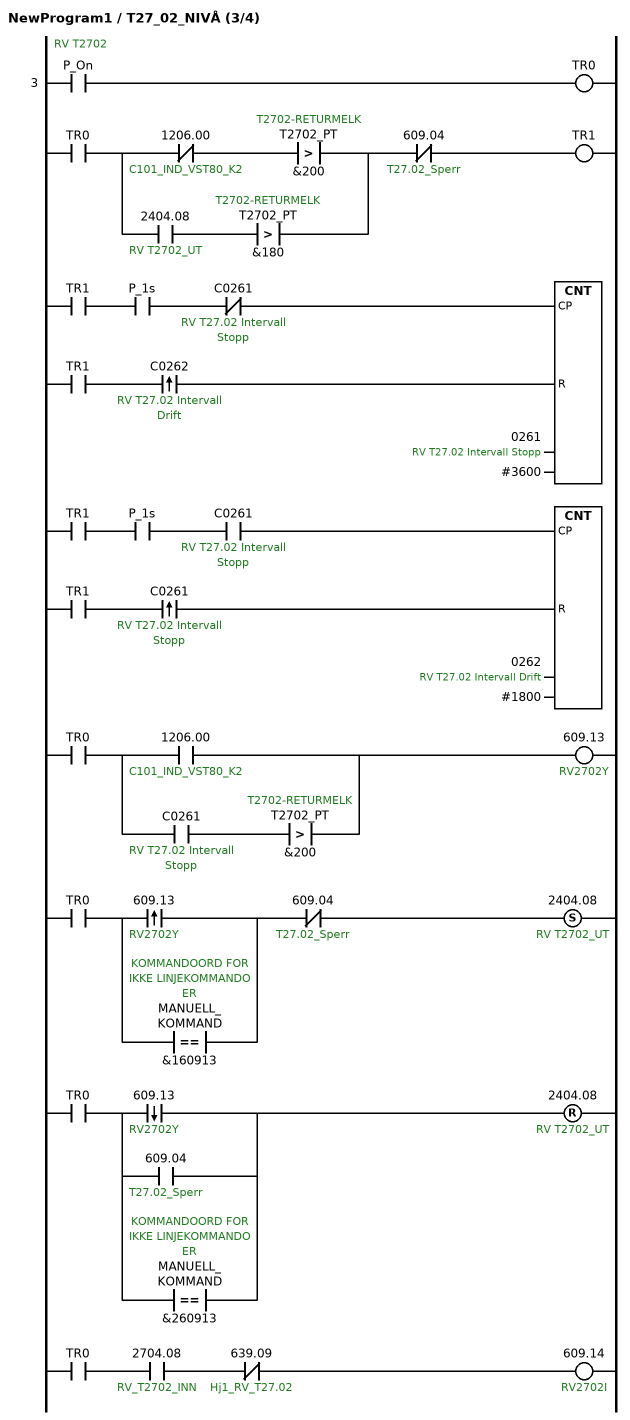
; [picture p984: NewProgram1 / T27_02_NIVÅ, rungs 3-3]
; rung 3: RV T2702
LD P_On
OUT TR0
LDNOT 1206.00  ; C101_IND_VST80_K2
AND>(320) T2702_PT &200  ; T2702-RETURMELK
LD 2404.08  ; RV T2702_UT
AND>(320) T2702_PT &180  ; T2702-RETURMELK
ORLD
ANDLD
ANDNOT 609.04  ; T27.02_Sperr
OUT TR1
AND P_1s
ANDNOT C0261  ; RV T27.02 Intervall Stopp
LD TR1
@AND C0262  ; RV T27.02 Intervall Drift
CNT 0261 #3600  ; RV T27.02 Intervall Stopp
LD TR1
AND P_1s
AND C0261  ; RV T27.02 Intervall Stopp
LD TR1
@AND C0261  ; RV T27.02 Intervall Stopp
CNT 0262 #1800  ; RV T27.02 Intervall Drift
LD TR0
LD 1206.00  ; C101_IND_VST80_K2
LD C0261  ; RV T27.02 Intervall Stopp
AND>(320) T2702_PT &200  ; T2702-RETURMELK
ORLD
ANDLD
OUT 609.13  ; RV2702Y
LD TR0
@LD 609.13  ; RV2702Y
OR=L(301) MANUELL_KOMMAND &160913  ; KOMMANDOORD FOR IKKE LINJEKOMMANDOER
ANDLD
ANDNOT 609.04  ; T27.02_Sperr
SET 2404.08  ; RV T2702_UT
LD TR0
%LD 609.13  ; RV2702Y
OR 609.04  ; T27.02_Sperr
OR=L(301) MANUELL_KOMMAND &260913  ; KOMMANDOORD FOR IKKE LINJEKOMMANDOER
ANDLD
RSET 2404.08  ; RV T2702_UT
LD TR0
AND 2704.08  ; RV_T2702_INN
ANDNOT 639.09  ; Hj1_RV_T27.02
OUT 609.14  ; RV2702I

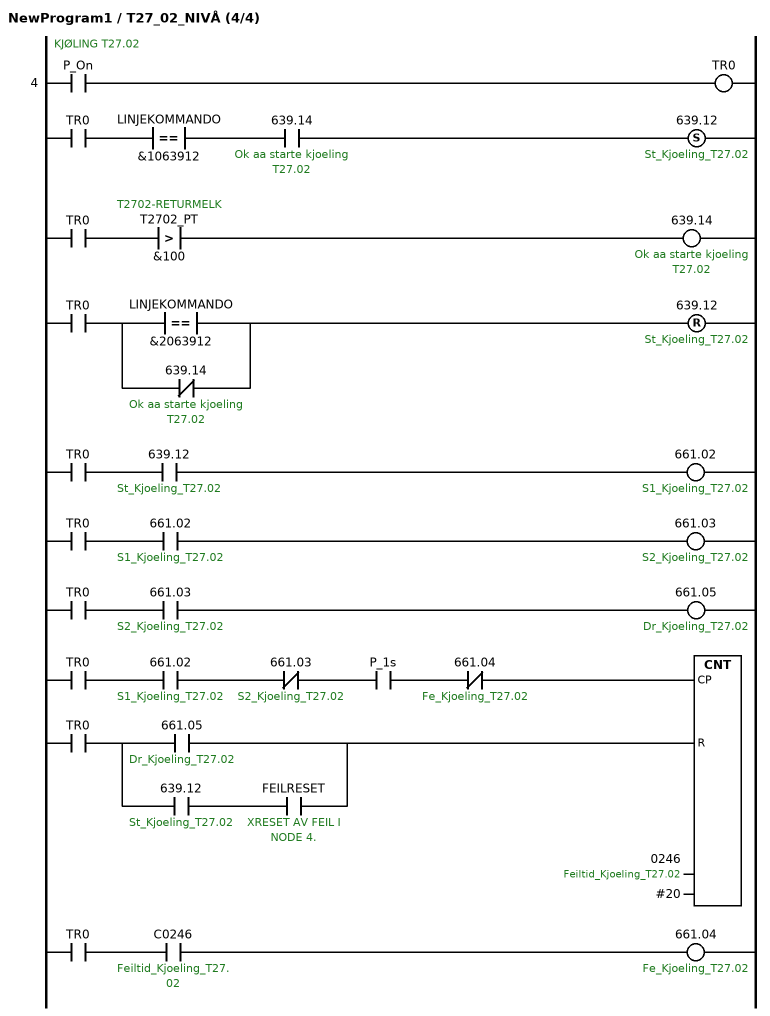
; rung 4: KJØLING T27.02
LD P_On
OUT TR0
AND=L(301) LINJEKOMMANDO &1063912
AND 639.14  ; Ok aa starte kjoeling T27.02
SET 639.12  ; St_Kjoeling_T27.02
LD TR0
AND>(320) T2702_PT &100  ; T2702-RETURMELK
OUT 639.14  ; Ok aa starte kjoeling T27.02
LD TR0
LD=L(301) LINJEKOMMANDO &2063912
ORNOT 639.14  ; Ok aa starte kjoeling T27.02
ANDLD
RSET 639.12  ; St_Kjoeling_T27.02
LD TR0
AND 639.12  ; St_Kjoeling_T27.02
OUT 661.02  ; S1_Kjoeling_T27.02
LD TR0
AND 661.02  ; S1_Kjoeling_T27.02
OUT 661.03  ; S2_Kjoeling_T27.02
LD TR0
AND 661.03  ; S2_Kjoeling_T27.02
OUT 661.05  ; Dr_Kjoeling_T27.02
LD TR0
AND 661.02  ; S1_Kjoeling_T27.02
ANDNOT 661.03  ; S2_Kjoeling_T27.02
AND P_1s
ANDNOT 661.04  ; Fe_Kjoeling_T27.02
LD TR0
LD 661.05  ; Dr_Kjoeling_T27.02
LD 639.12  ; St_Kjoeling_T27.02
AND FEILRESET  ; XRESET AV FEIL I NODE 4.
ORLD
ANDLD
CNT 0246 #20  ; Feiltid_Kjoeling_T27.02
LD TR0
AND C0246  ; Feiltid_Kjoeling_T27.02
OUT 661.04  ; Fe_Kjoeling_T27.02

### Section T27_02

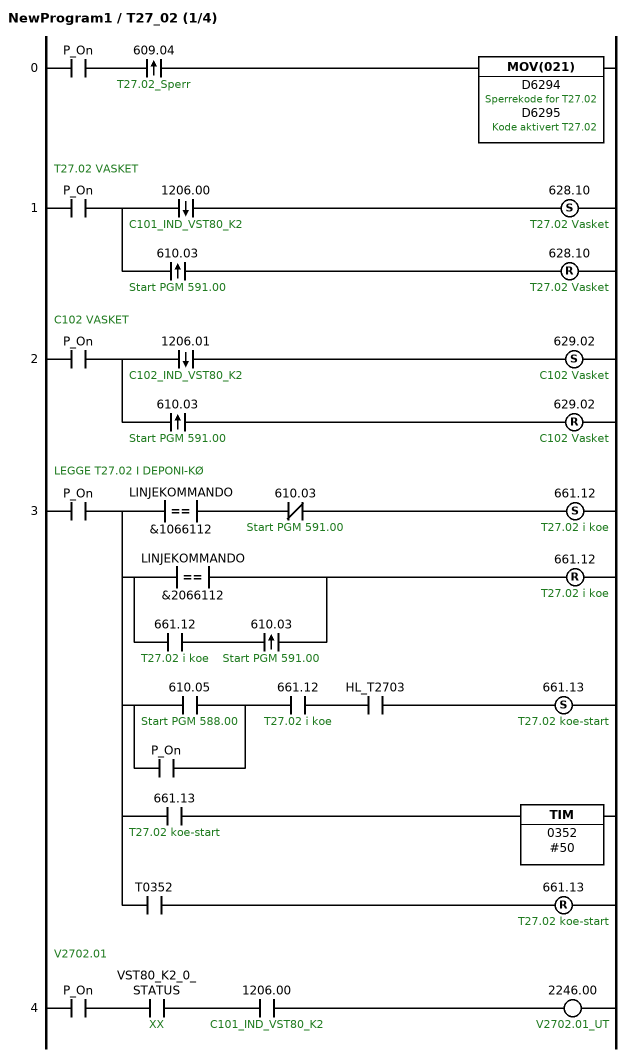
; rung 0
LD P_On
@AND 609.04  ; T27.02_Sperr
MOV(021) D6294 D6295  ; Sperrekode for T27.02, Kode aktivert T27.02
; rung 1: T27.02 VASKET
LD P_On
OUT TR0
%AND 1206.00  ; C101_IND_VST80_K2
SET 628.10  ; T27.02 Vasket
LD TR0
@AND 610.03  ; Start PGM 591.00
RSET 628.10  ; T27.02 Vasket
; rung 2: C102 VASKET
LD P_On
OUT TR0
%AND 1206.01  ; C102_IND_VST80_K2
SET 629.02  ; C102 Vasket
LD TR0
@AND 610.03  ; Start PGM 591.00
RSET 629.02  ; C102 Vasket
; rung 3: LEGGE T27.02 I DEPONI-KØ
LD P_On
OUT TR0
AND=L(301) LINJEKOMMANDO &1066112
ANDNOT 610.03  ; Start PGM 591.00
SET 661.12  ; T27.02 i koe
LD TR0
LD=L(301) LINJEKOMMANDO &2066112
LD 661.12  ; T27.02 i koe
@AND 610.03  ; Start PGM 591.00
ORLD
ANDLD
RSET 661.12  ; T27.02 i koe
LD TR0
LD 610.05  ; Start PGM 588.00
OR P_On
ANDLD
AND 661.12  ; T27.02 i koe
AND HL_T2703
SET 661.13  ; T27.02 koe-start
LD TR0
AND 661.13  ; T27.02 koe-start
TIM 0352 #50
LD TR0
AND T0352
RSET 661.13  ; T27.02 koe-start
; rung 4: V2702.01
LD P_On
AND VST80_K2_0_STATUS  ; XX
AND 1206.00  ; C101_IND_VST80_K2
OUT 2246.00  ; V2702.01_UT

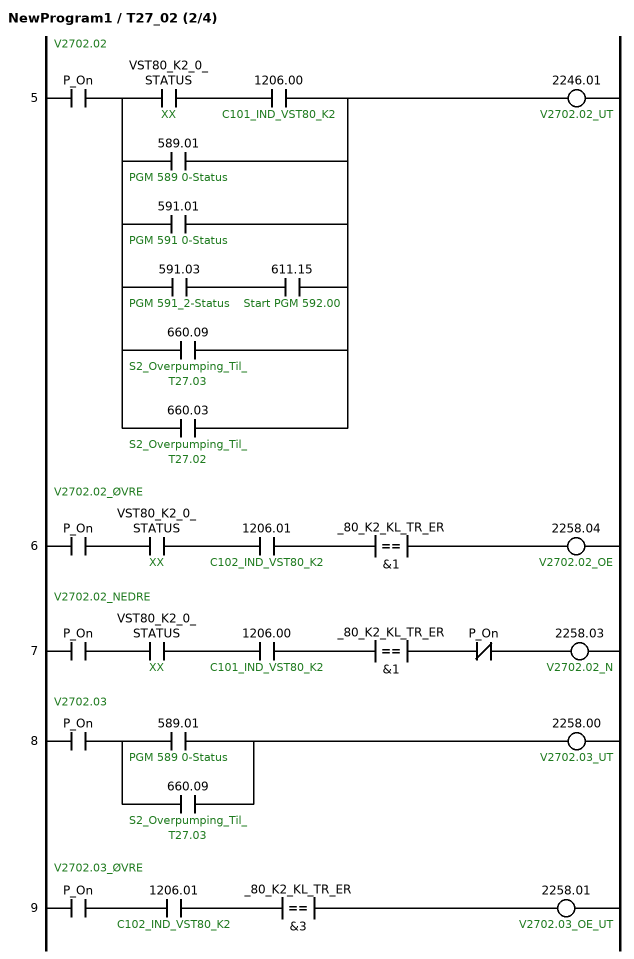
; rung 5: V2702.02
LD P_On
LD VST80_K2_0_STATUS  ; XX
AND 1206.00  ; C101_IND_VST80_K2
OR 589.01  ; PGM 589 0-Status
OR 591.01  ; PGM 591 0-Status
LD 591.03  ; PGM 591_2-Status
AND 611.15  ; Start PGM 592.00
ORLD
OR 660.09  ; S2_Overpumping_Til_T27.03
OR 660.03  ; S2_Overpumping_Til_T27.02
ANDLD
OUT 2246.01  ; V2702.02_UT
; rung 6: V2702.02_ØVRE
LD P_On
AND VST80_K2_0_STATUS  ; XX
AND 1206.01  ; C102_IND_VST80_K2
AND=(300) _80_K2_KL_TR_ER &1
OUT 2258.04  ; V2702.02_OE
; rung 7: V2702.02_NEDRE
LD P_On
AND VST80_K2_0_STATUS  ; XX
AND 1206.00  ; C101_IND_VST80_K2
AND=(300) _80_K2_KL_TR_ER &1
ANDNOT P_On
OUT 2258.03  ; V2702.02_N
; rung 8: V2702.03
LD P_On
LD 589.01  ; PGM 589 0-Status
OR 660.09  ; S2_Overpumping_Til_T27.03
ANDLD
OUT 2258.00  ; V2702.03_UT
; rung 9: V2702.03_ØVRE
LD P_On
AND 1206.01  ; C102_IND_VST80_K2
AND=(300) _80_K2_KL_TR_ER &3
OUT 2258.01  ; V2702.03_OE_UT

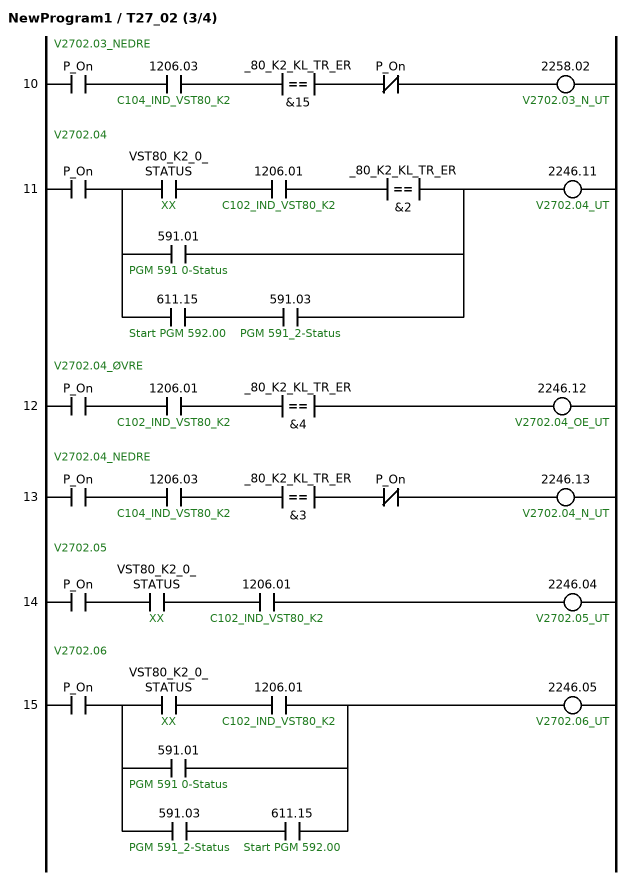
; rung 10: V2702.03_NEDRE
LD P_On
AND 1206.03  ; C104_IND_VST80_K2
AND=(300) _80_K2_KL_TR_ER &15
ANDNOT P_On
OUT 2258.02  ; V2702.03_N_UT
; rung 11: V2702.04
LD P_On
LD VST80_K2_0_STATUS  ; XX
AND 1206.01  ; C102_IND_VST80_K2
AND=(300) _80_K2_KL_TR_ER &2
OR 591.01  ; PGM 591 0-Status
LD 611.15  ; Start PGM 592.00
AND 591.03  ; PGM 591_2-Status
ORLD
ANDLD
OUT 2246.11  ; V2702.04_UT
; rung 12: V2702.04_ØVRE
LD P_On
AND 1206.01  ; C102_IND_VST80_K2
AND=(300) _80_K2_KL_TR_ER &4
OUT 2246.12  ; V2702.04_OE_UT
; rung 13: V2702.04_NEDRE
LD P_On
AND 1206.03  ; C104_IND_VST80_K2
AND=(300) _80_K2_KL_TR_ER &3
ANDNOT P_On
OUT 2246.13  ; V2702.04_N_UT
; rung 14: V2702.05
LD P_On
AND VST80_K2_0_STATUS  ; XX
AND 1206.01  ; C102_IND_VST80_K2
OUT 2246.04  ; V2702.05_UT
; rung 15: V2702.06
LD P_On
LD VST80_K2_0_STATUS  ; XX
AND 1206.01  ; C102_IND_VST80_K2
OR 591.01  ; PGM 591 0-Status
LD 591.03  ; PGM 591_2-Status
AND 611.15  ; Start PGM 592.00
ORLD
ANDLD
OUT 2246.05  ; V2702.06_UT

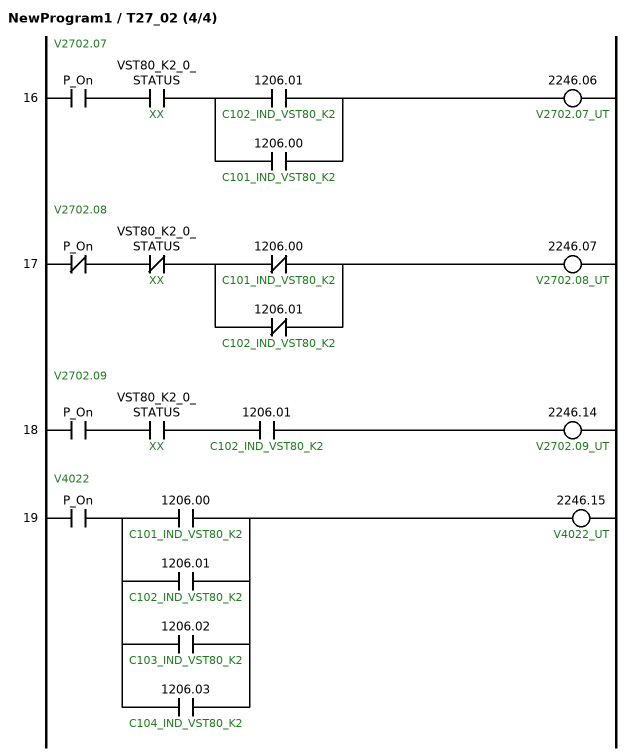
; rung 16: V2702.07
LD P_On
AND VST80_K2_0_STATUS  ; XX
LD 1206.01  ; C102_IND_VST80_K2
OR 1206.00  ; C101_IND_VST80_K2
ANDLD
OUT 2246.06  ; V2702.07_UT
; rung 17: V2702.08
LDNOT P_On
ANDNOT VST80_K2_0_STATUS  ; XX
LDNOT 1206.00  ; C101_IND_VST80_K2
ORNOT 1206.01  ; C102_IND_VST80_K2
ANDLD
OUT 2246.07  ; V2702.08_UT
; rung 18: V2702.09
LD P_On
AND VST80_K2_0_STATUS  ; XX
AND 1206.01  ; C102_IND_VST80_K2
OUT 2246.14  ; V2702.09_UT
; rung 19: V4022
LD P_On
LD 1206.00  ; C101_IND_VST80_K2
OR 1206.01  ; C102_IND_VST80_K2
OR 1206.02  ; C103_IND_VST80_K2
OR 1206.03  ; C104_IND_VST80_K2
ANDLD
OUT 2246.15  ; V4022_UT

### Section T27_03_SPERR

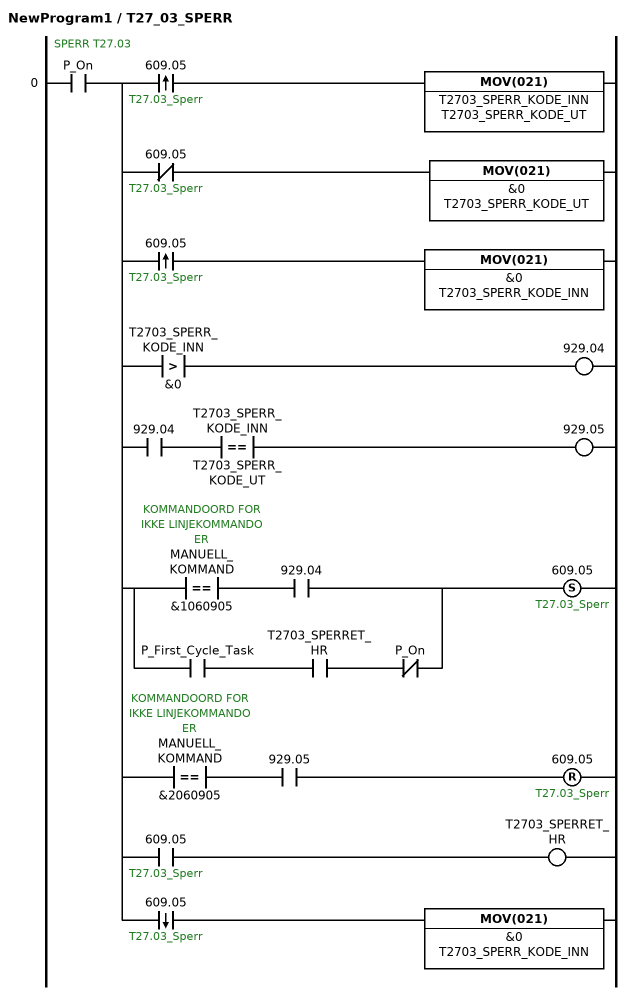
; rung 0: SPERR T27.03
LD P_On
OUT TR0
@AND 609.05  ; T27.03_Sperr
MOV(021) T2703_SPERR_KODE_INN T2703_SPERR_KODE_UT
LD TR0
ANDNOT 609.05  ; T27.03_Sperr
MOV(021) &0 T2703_SPERR_KODE_UT
LD TR0
@AND 609.05  ; T27.03_Sperr
MOV(021) &0 T2703_SPERR_KODE_INN
LD TR0
AND>(320) T2703_SPERR_KODE_INN &0
OUT 929.04
LD TR0
AND 929.04
AND=(300) T2703_SPERR_KODE_INN T2703_SPERR_KODE_UT
OUT 929.05
LD TR0
LD=L(301) MANUELL_KOMMAND &1060905  ; KOMMANDOORD FOR IKKE LINJEKOMMANDOER
AND 929.04
LD P_First_Cycle_Task
AND T2703_SPERRET_HR
ANDNOT P_On
ORLD
ANDLD
SET 609.05  ; T27.03_Sperr
LD TR0
AND=L(301) MANUELL_KOMMAND &2060905  ; KOMMANDOORD FOR IKKE LINJEKOMMANDOER
AND 929.05
RSET 609.05  ; T27.03_Sperr
LD TR0
AND 609.05  ; T27.03_Sperr
OUT T2703_SPERRET_HR
LD TR0
%AND 609.05  ; T27.03_Sperr
MOV(021) &0 T2703_SPERR_KODE_INN

### Section T27_03_NIVÅ

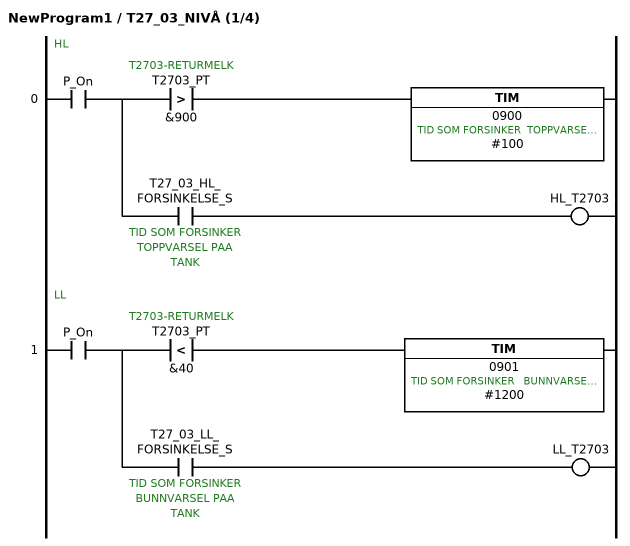
; rung 0: HL
LD P_On
OUT TR0
AND>(320) T2703_PT &900  ; T2703-RETURMELK
TIM 0900 #100  ; TID SOM FORSINKER  TOPPVARSEL PAA  TANK
LD TR0
AND T27_03_HL_FORSINKELSE_S  ; TID SOM FORSINKER  TOPPVARSEL PAA  TANK
OUT HL_T2703
; rung 1: LL
LD P_On
OUT TR0
AND<(310) T2703_PT &40  ; T2703-RETURMELK
TIM 0901 #1200  ; TID SOM FORSINKER   BUNNVARSEL PAA TANK
LD TR0
AND T27_03_LL_FORSINKELSE_S  ; TID SOM FORSINKER   BUNNVARSEL PAA TANK
OUT LL_T2703

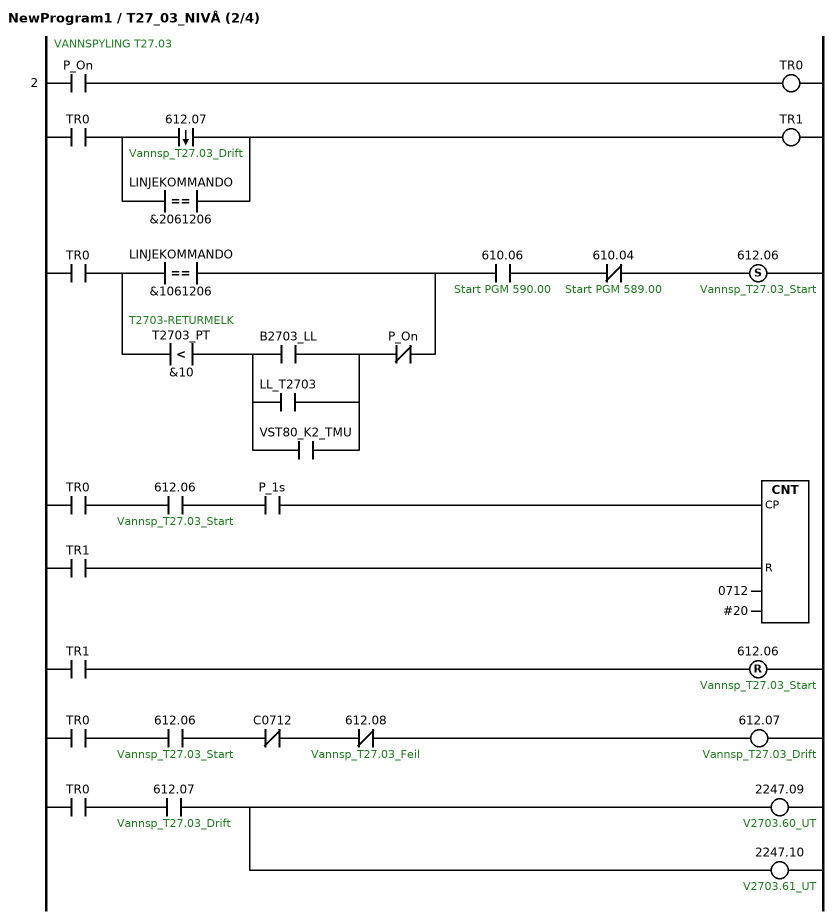
; rung 2: VANNSPYLING T27.03
LD P_On
OUT TR0
LD=L(301) LINJEKOMMANDO &1061206
LD<(310) T2703_PT &10  ; T2703-RETURMELK
LD B2703_LL
OR LL_T2703
OR VST80_K2_TMU
ANDLD
ANDNOT P_On
ORLD
ANDLD
AND 610.06  ; Start PGM 590.00
ANDNOT 610.04  ; Start PGM 589.00
SET 612.06  ; Vannsp_T27.03_Start
LD TR0
AND 612.06  ; Vannsp_T27.03_Start
AND P_1s
LD TR0
%LD 612.07  ; Vannsp_T27.03_Drift
OR=L(301) LINJEKOMMANDO &2061206
ANDLD
OUT TR1
CNT 0712 #20
LD TR1
RSET 612.06  ; Vannsp_T27.03_Start
LD TR0
AND 612.06  ; Vannsp_T27.03_Start
ANDNOT C0712
ANDNOT 612.08  ; Vannsp_T27.03_Feil
OUT 612.07  ; Vannsp_T27.03_Drift
LD TR0
AND 612.07  ; Vannsp_T27.03_Drift
OUT 2247.09  ; V2703.60_UT
OUT 2247.10  ; V2703.61_UT

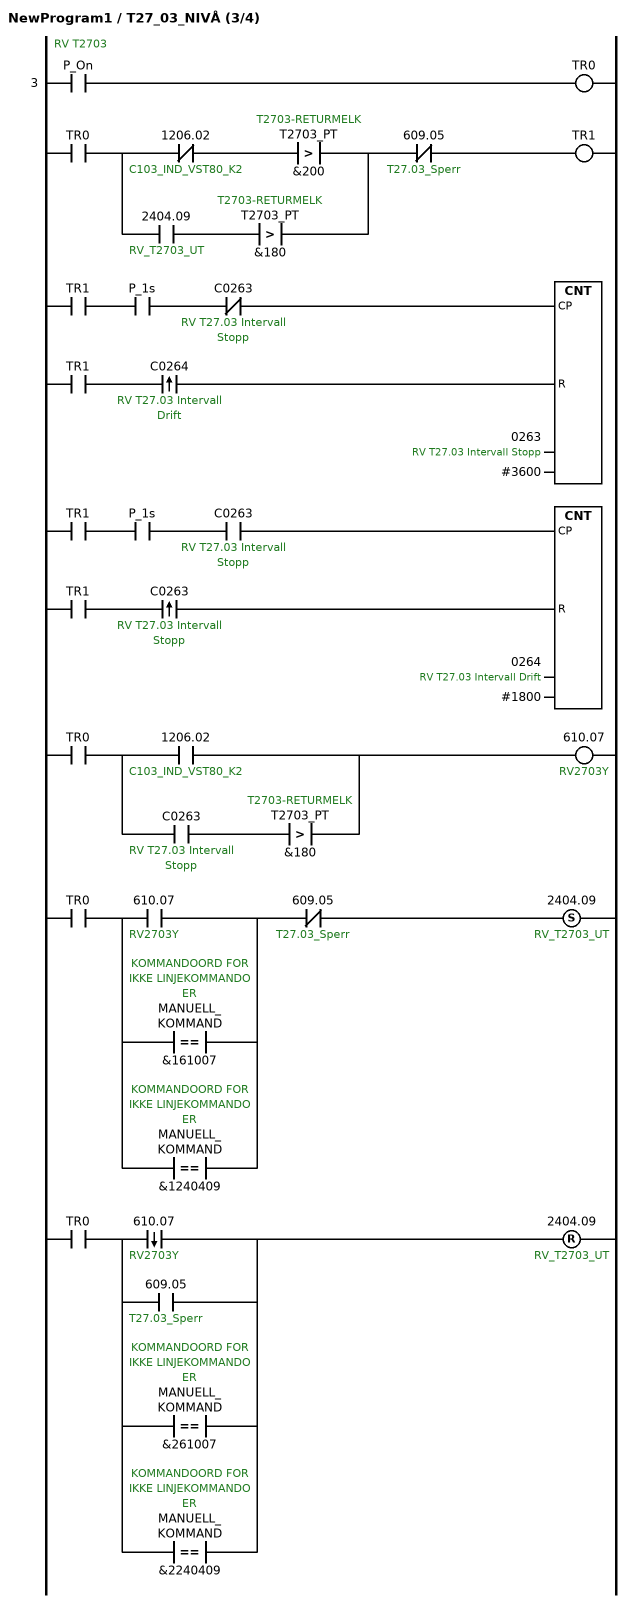
; rung 3: RV T2703
LD P_On
OUT TR0
LDNOT 1206.02  ; C103_IND_VST80_K2
AND>(320) T2703_PT &200  ; T2703-RETURMELK
LD 2404.09  ; RV_T2703_UT
AND>(320) T2703_PT &180  ; T2703-RETURMELK
ORLD
ANDLD
ANDNOT 609.05  ; T27.03_Sperr
OUT TR1
AND P_1s
ANDNOT C0263  ; RV T27.03 Intervall Stopp
LD TR1
@AND C0264  ; RV T27.03 Intervall Drift
CNT 0263 #3600  ; RV T27.03 Intervall Stopp
LD TR1
AND P_1s
AND C0263  ; RV T27.03 Intervall Stopp
LD TR1
@AND C0263  ; RV T27.03 Intervall Stopp
CNT 0264 #1800  ; RV T27.03 Intervall Drift
LD TR0
LD 1206.02  ; C103_IND_VST80_K2
LD C0263  ; RV T27.03 Intervall Stopp
AND>(320) T2703_PT &180  ; T2703-RETURMELK
ORLD
ANDLD
OUT 610.07  ; RV2703Y
LD TR0
LD 610.07  ; RV2703Y
OR=L(301) MANUELL_KOMMAND &161007  ; KOMMANDOORD FOR IKKE LINJEKOMMANDOER
OR=L(301) MANUELL_KOMMAND &1240409  ; KOMMANDOORD FOR IKKE LINJEKOMMANDOER
ANDLD
ANDNOT 609.05  ; T27.03_Sperr
SET 2404.09  ; RV_T2703_UT
LD TR0
%LD 610.07  ; RV2703Y
OR 609.05  ; T27.03_Sperr
OR=L(301) MANUELL_KOMMAND &261007  ; KOMMANDOORD FOR IKKE LINJEKOMMANDOER
OR=L(301) MANUELL_KOMMAND &2240409  ; KOMMANDOORD FOR IKKE LINJEKOMMANDOER
ANDLD
RSET 2404.09  ; RV_T2703_UT

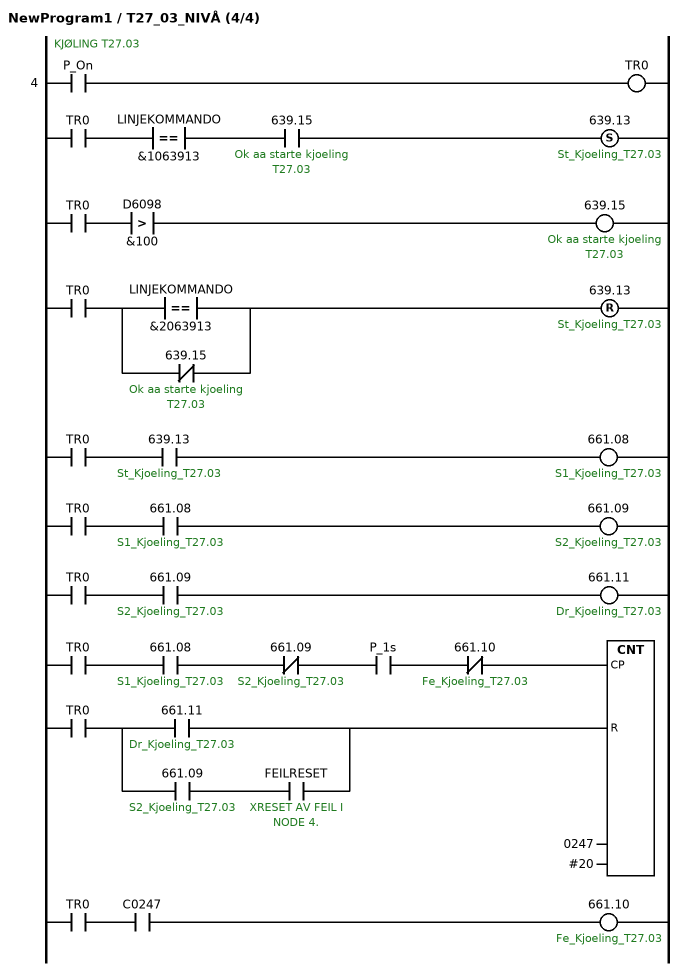
; rung 4: KJØLING T27.03
LD P_On
OUT TR0
AND=L(301) LINJEKOMMANDO &1063913
AND 639.15  ; Ok aa starte kjoeling T27.03
SET 639.13  ; St_Kjoeling_T27.03
LD TR0
AND>(320) D6098 &100
OUT 639.15  ; Ok aa starte kjoeling T27.03
LD TR0
LD=L(301) LINJEKOMMANDO &2063913
ORNOT 639.15  ; Ok aa starte kjoeling T27.03
ANDLD
RSET 639.13  ; St_Kjoeling_T27.03
LD TR0
AND 639.13  ; St_Kjoeling_T27.03
OUT 661.08  ; S1_Kjoeling_T27.03
LD TR0
AND 661.08  ; S1_Kjoeling_T27.03
OUT 661.09  ; S2_Kjoeling_T27.03
LD TR0
AND 661.09  ; S2_Kjoeling_T27.03
OUT 661.11  ; Dr_Kjoeling_T27.03
LD TR0
AND 661.08  ; S1_Kjoeling_T27.03
ANDNOT 661.09  ; S2_Kjoeling_T27.03
AND P_1s
ANDNOT 661.10  ; Fe_Kjoeling_T27.03
LD TR0
LD 661.11  ; Dr_Kjoeling_T27.03
LD 661.09  ; S2_Kjoeling_T27.03
AND FEILRESET  ; XRESET AV FEIL I NODE 4.
ORLD
ANDLD
CNT 0247 #20
LD TR0
AND C0247
OUT 661.10  ; Fe_Kjoeling_T27.03

### Section T27_03

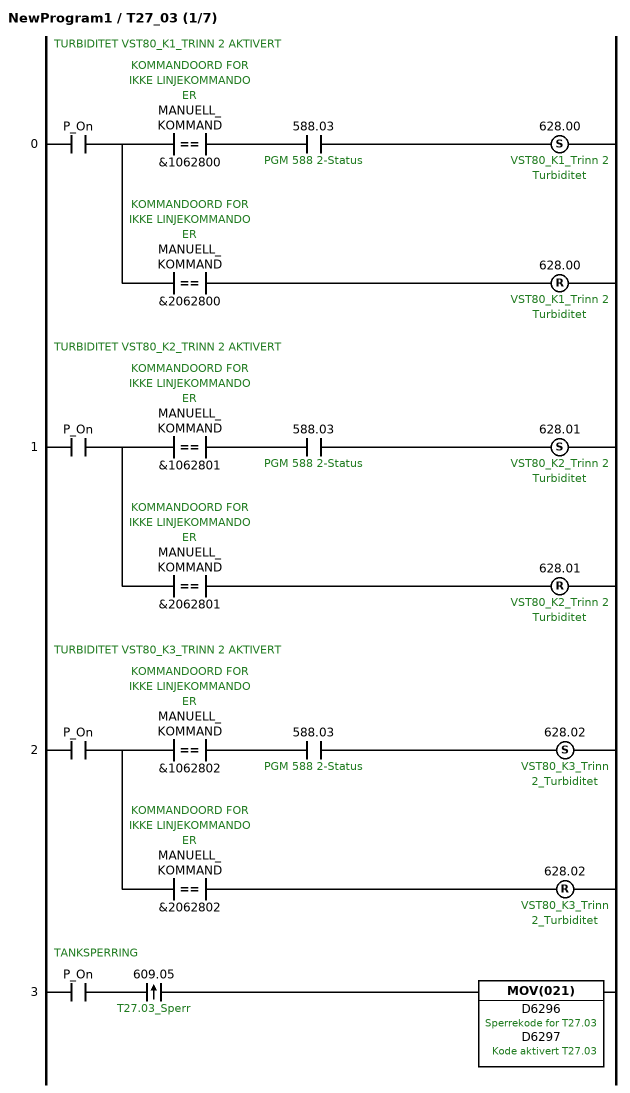
; rung 0: TURBIDITET VST80_K1_TRINN 2 AKTIVERT
LD P_On
OUT TR0
AND=L(301) MANUELL_KOMMAND &1062800  ; KOMMANDOORD FOR IKKE LINJEKOMMANDOER
AND 588.03  ; PGM 588 2-Status
SET 628.00  ; VST80_K1_Trinn 2 Turbiditet
LD TR0
AND=L(301) MANUELL_KOMMAND &2062800  ; KOMMANDOORD FOR IKKE LINJEKOMMANDOER
RSET 628.00  ; VST80_K1_Trinn 2 Turbiditet
; rung 1: TURBIDITET VST80_K2_TRINN 2 AKTIVERT
LD P_On
OUT TR0
AND=L(301) MANUELL_KOMMAND &1062801  ; KOMMANDOORD FOR IKKE LINJEKOMMANDOER
AND 588.03  ; PGM 588 2-Status
SET 628.01  ; VST80_K2_Trinn 2 Turbiditet
LD TR0
AND=L(301) MANUELL_KOMMAND &2062801  ; KOMMANDOORD FOR IKKE LINJEKOMMANDOER
RSET 628.01  ; VST80_K2_Trinn 2 Turbiditet
; rung 2: TURBIDITET VST80_K3_TRINN 2 AKTIVERT
LD P_On
OUT TR0
AND=L(301) MANUELL_KOMMAND &1062802  ; KOMMANDOORD FOR IKKE LINJEKOMMANDOER
AND 588.03  ; PGM 588 2-Status
SET 628.02  ; VST80_K3_Trinn 2_Turbiditet
LD TR0
AND=L(301) MANUELL_KOMMAND &2062802  ; KOMMANDOORD FOR IKKE LINJEKOMMANDOER
RSET 628.02  ; VST80_K3_Trinn 2_Turbiditet
; rung 3: TANKSPERRING
LD P_On
@AND 609.05  ; T27.03_Sperr
MOV(021) D6296 D6297  ; Sperrekode for T27.03, Kode aktivert T27.03

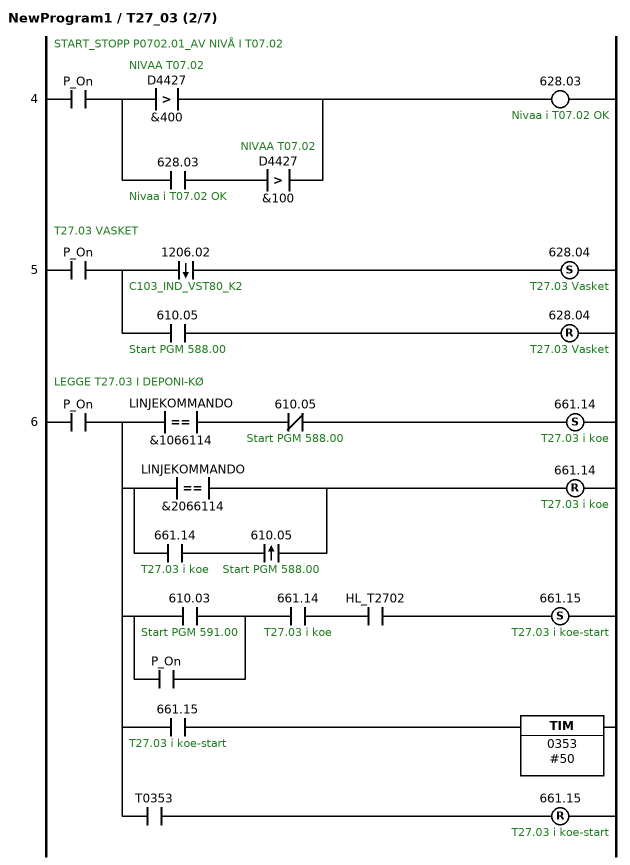
; rung 4: START_STOPP P0702.01_AV NIVÅ I T07.02
LD P_On
LD>(320) D4427 &400  ; NIVAA T07.02
LD 628.03  ; Nivaa i T07.02 OK
AND>(320) D4427 &100  ; NIVAA T07.02
ORLD
ANDLD
OUT 628.03  ; Nivaa i T07.02 OK
; rung 5: T27.03 VASKET
LD P_On
OUT TR0
%AND 1206.02  ; C103_IND_VST80_K2
SET 628.04  ; T27.03 Vasket
LD TR0
AND 610.05  ; Start PGM 588.00
RSET 628.04  ; T27.03 Vasket
; rung 6: LEGGE T27.03 I DEPONI-KØ
LD P_On
OUT TR0
AND=L(301) LINJEKOMMANDO &1066114
ANDNOT 610.05  ; Start PGM 588.00
SET 661.14  ; T27.03 i koe
LD TR0
LD=L(301) LINJEKOMMANDO &2066114
LD 661.14  ; T27.03 i koe
@AND 610.05  ; Start PGM 588.00
ORLD
ANDLD
RSET 661.14  ; T27.03 i koe
LD TR0
LD 610.03  ; Start PGM 591.00
OR P_On
ANDLD
AND 661.14  ; T27.03 i koe
AND HL_T2702
SET 661.15  ; T27.03 i koe-start
LD TR0
AND 661.15  ; T27.03 i koe-start
TIM 0353 #50
LD TR0
AND T0353
RSET 661.15  ; T27.03 i koe-start

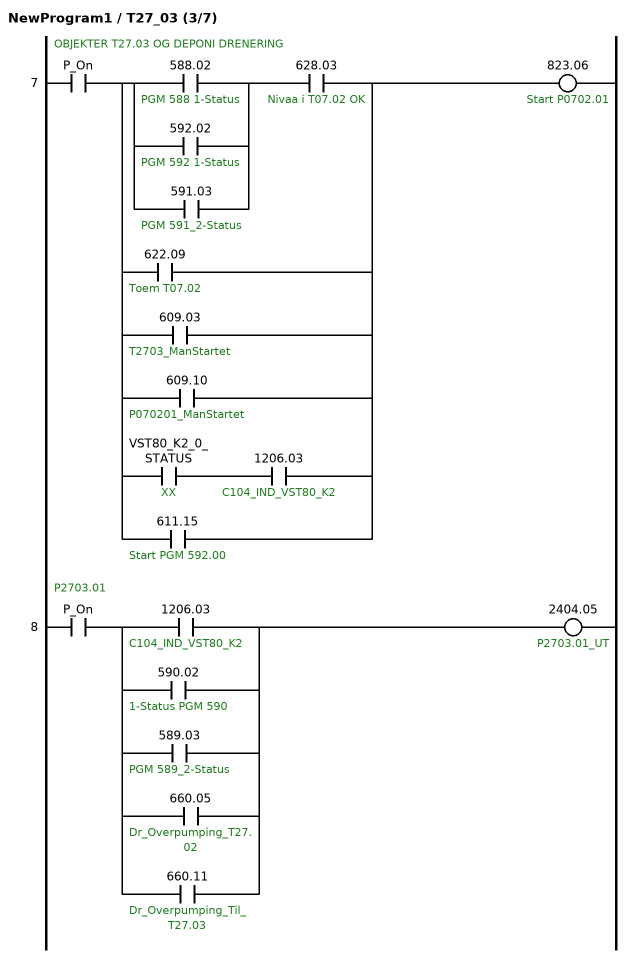
; rung 7: OBJEKTER T27.03 OG DEPONI DRENERING
LD P_On
LD 588.02  ; PGM 588 1-Status
OR 592.02  ; PGM 592 1-Status
OR 591.03  ; PGM 591_2-Status
AND 628.03  ; Nivaa i T07.02 OK
OR 622.09  ; Toem T07.02
OR 609.03  ; T2703_ManStartet
OR 609.10  ; P070201_ManStartet
LD VST80_K2_0_STATUS  ; XX
AND 1206.03  ; C104_IND_VST80_K2
ORLD
OR 611.15  ; Start PGM 592.00
ANDLD
OUT 823.06  ; Start P0702.01
; rung 8: P2703.01
LD P_On
LD 1206.03  ; C104_IND_VST80_K2
OR 590.02  ; 1-Status PGM 590
OR 589.03  ; PGM 589_2-Status
OR 660.05  ; Dr_Overpumping_T27.02
OR 660.11  ; Dr_Overpumping_Til_T27.03
ANDLD
OUT 2404.05  ; P2703.01_UT

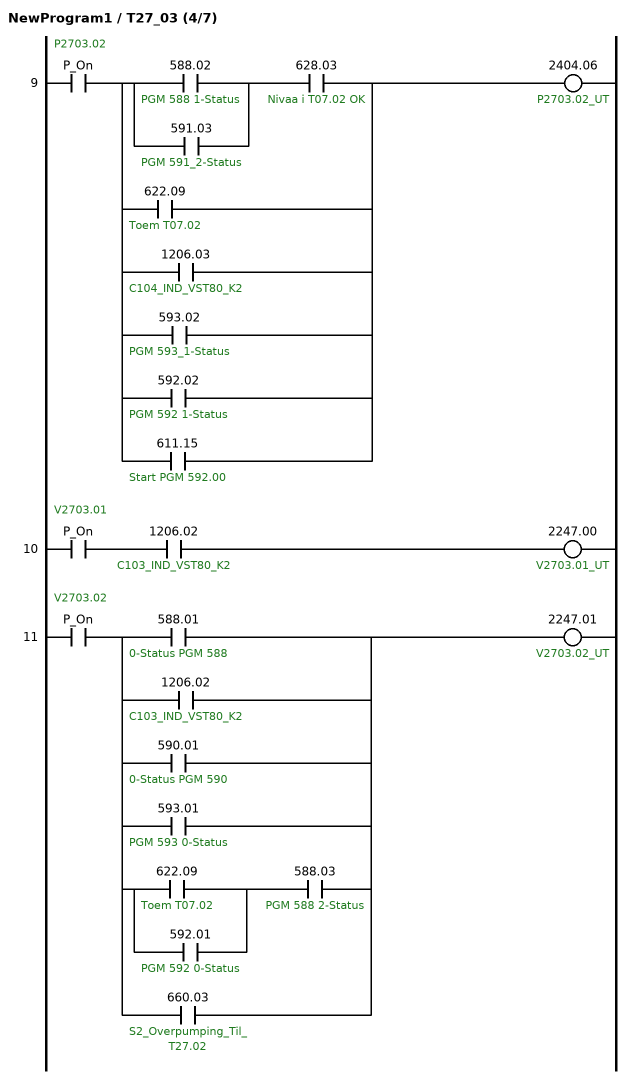
; rung 9: P2703.02
LD P_On
LD 588.02  ; PGM 588 1-Status
OR 591.03  ; PGM 591_2-Status
AND 628.03  ; Nivaa i T07.02 OK
OR 622.09  ; Toem T07.02
OR 1206.03  ; C104_IND_VST80_K2
OR 593.02  ; PGM 593_1-Status
OR 592.02  ; PGM 592 1-Status
OR 611.15  ; Start PGM 592.00
ANDLD
OUT 2404.06  ; P2703.02_UT
; rung 10: V2703.01
LD P_On
AND 1206.02  ; C103_IND_VST80_K2
OUT 2247.00  ; V2703.01_UT
; rung 11: V2703.02
LD P_On
LD 588.01  ; 0-Status PGM 588
OR 1206.02  ; C103_IND_VST80_K2
OR 590.01  ; 0-Status PGM 590
OR 593.01  ; PGM 593 0-Status
LD 622.09  ; Toem T07.02
OR 592.01  ; PGM 592 0-Status
AND 588.03  ; PGM 588 2-Status
ORLD
OR 660.03  ; S2_Overpumping_Til_T27.02
ANDLD
OUT 2247.01  ; V2703.02_UT

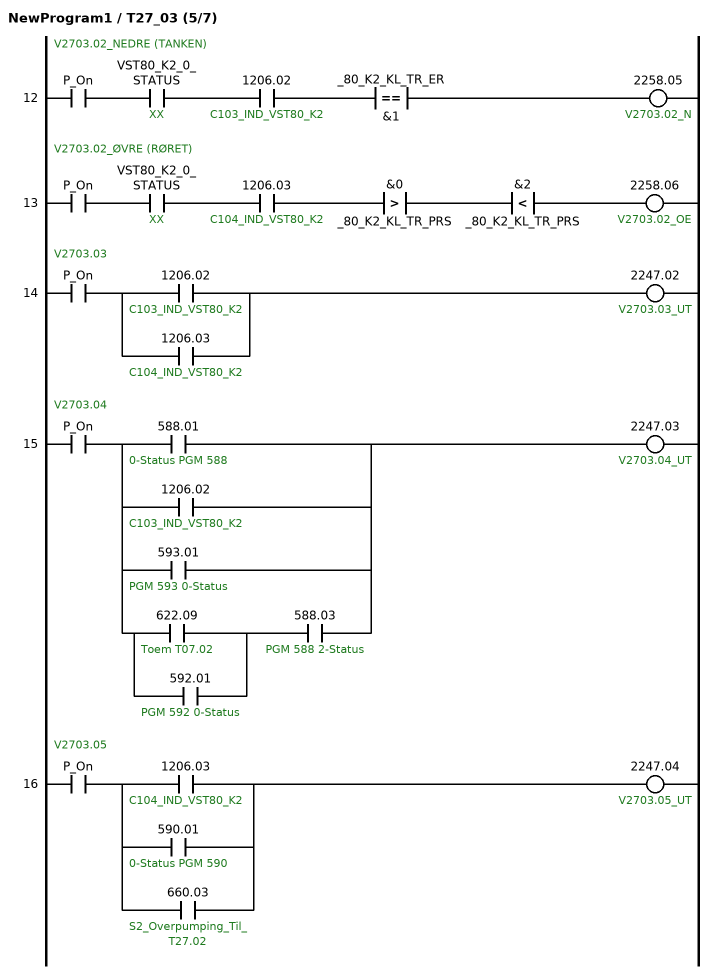
; rung 12: V2703.02_NEDRE (TANKEN)
LD P_On
AND VST80_K2_0_STATUS  ; XX
AND 1206.02  ; C103_IND_VST80_K2
AND=(300) _80_K2_KL_TR_ER &1
OUT 2258.05  ; V2703.02_N
; rung 13: V2703.02_ØVRE (RØRET)
LD P_On
AND VST80_K2_0_STATUS  ; XX
AND 1206.03  ; C104_IND_VST80_K2
AND>(320) &0 _80_K2_KL_TR_PRS
AND<(310) &2 _80_K2_KL_TR_PRS
OUT 2258.06  ; V2703.02_OE
; rung 14: V2703.03
LD P_On
LD 1206.02  ; C103_IND_VST80_K2
OR 1206.03  ; C104_IND_VST80_K2
ANDLD
OUT 2247.02  ; V2703.03_UT
; rung 15: V2703.04
LD P_On
LD 588.01  ; 0-Status PGM 588
OR 1206.02  ; C103_IND_VST80_K2
OR 593.01  ; PGM 593 0-Status
LD 622.09  ; Toem T07.02
OR 592.01  ; PGM 592 0-Status
AND 588.03  ; PGM 588 2-Status
ORLD
ANDLD
OUT 2247.03  ; V2703.04_UT
; rung 16: V2703.05
LD P_On
LD 1206.03  ; C104_IND_VST80_K2
OR 590.01  ; 0-Status PGM 590
OR 660.03  ; S2_Overpumping_Til_T27.02
ANDLD
OUT 2247.04  ; V2703.05_UT

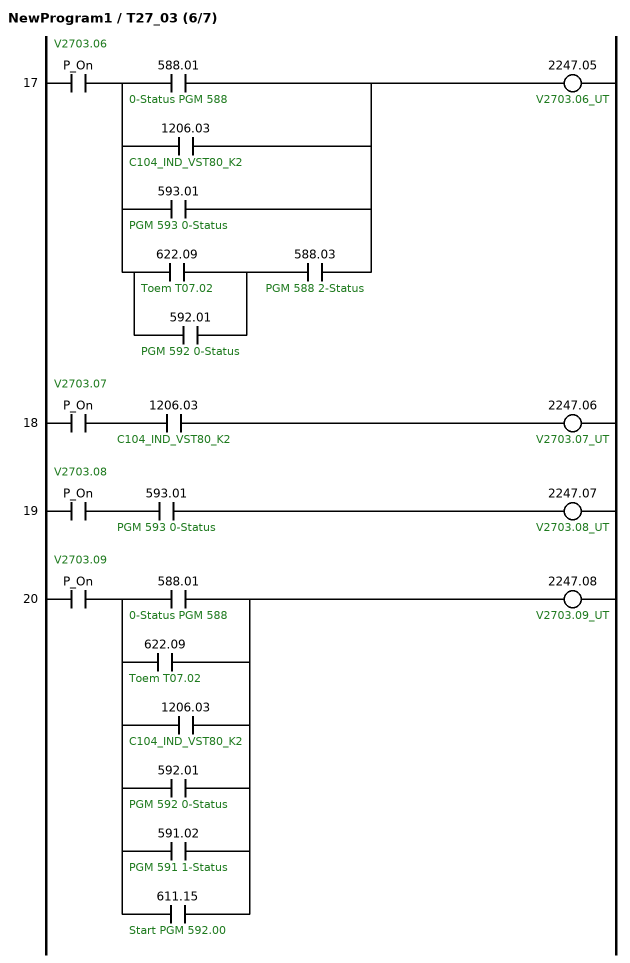
; rung 17: V2703.06
LD P_On
LD 588.01  ; 0-Status PGM 588
OR 1206.03  ; C104_IND_VST80_K2
OR 593.01  ; PGM 593 0-Status
LD 622.09  ; Toem T07.02
OR 592.01  ; PGM 592 0-Status
AND 588.03  ; PGM 588 2-Status
ORLD
ANDLD
OUT 2247.05  ; V2703.06_UT
; rung 18: V2703.07
LD P_On
AND 1206.03  ; C104_IND_VST80_K2
OUT 2247.06  ; V2703.07_UT
; rung 19: V2703.08
LD P_On
AND 593.01  ; PGM 593 0-Status
OUT 2247.07  ; V2703.08_UT
; rung 20: V2703.09
LD P_On
LD 588.01  ; 0-Status PGM 588
OR 622.09  ; Toem T07.02
OR 1206.03  ; C104_IND_VST80_K2
OR 592.01  ; PGM 592 0-Status
OR 591.02  ; PGM 591 1-Status
OR 611.15  ; Start PGM 592.00
ANDLD
OUT 2247.08  ; V2703.09_UT

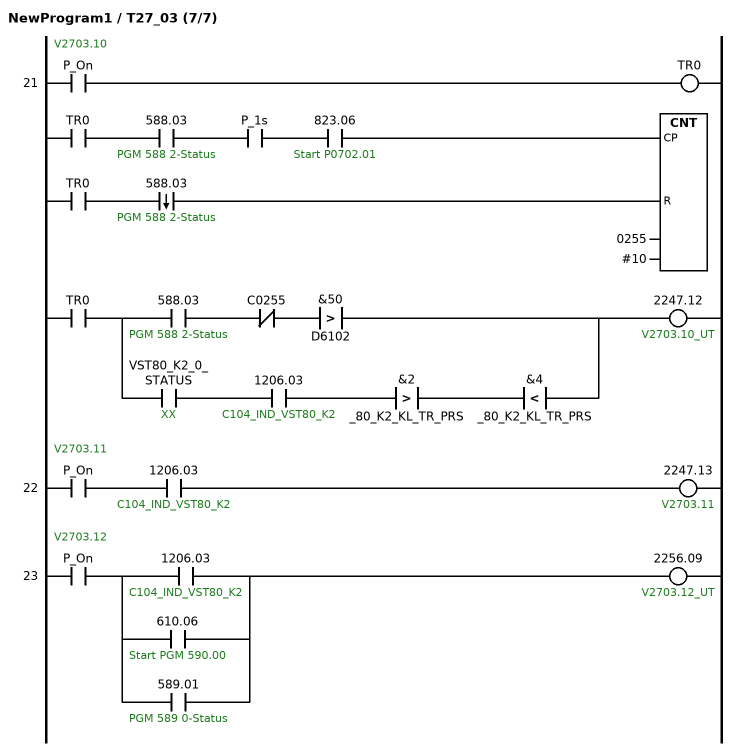
; rung 21: V2703.10
LD P_On
OUT TR0
AND 588.03  ; PGM 588 2-Status
AND P_1s
AND 823.06  ; Start P0702.01
LD TR0
%AND 588.03  ; PGM 588 2-Status
CNT 0255 #10
LD TR0
LD 588.03  ; PGM 588 2-Status
ANDNOT C0255
AND>(320) &50 D6102
LD VST80_K2_0_STATUS  ; XX
AND 1206.03  ; C104_IND_VST80_K2
AND>(320) &2 _80_K2_KL_TR_PRS
AND<(310) &4 _80_K2_KL_TR_PRS
ORLD
ANDLD
OUT 2247.12  ; V2703.10_UT
; rung 22: V2703.11
LD P_On
AND 1206.03  ; C104_IND_VST80_K2
OUT 2247.13  ; V2703.11
; rung 23: V2703.12
LD P_On
LD 1206.03  ; C104_IND_VST80_K2
OR 610.06  ; Start PGM 590.00
OR 589.01  ; PGM 589 0-Status
ANDLD
OUT 2256.09  ; V2703.12_UT

### Section P8024_RETUR_C07_08

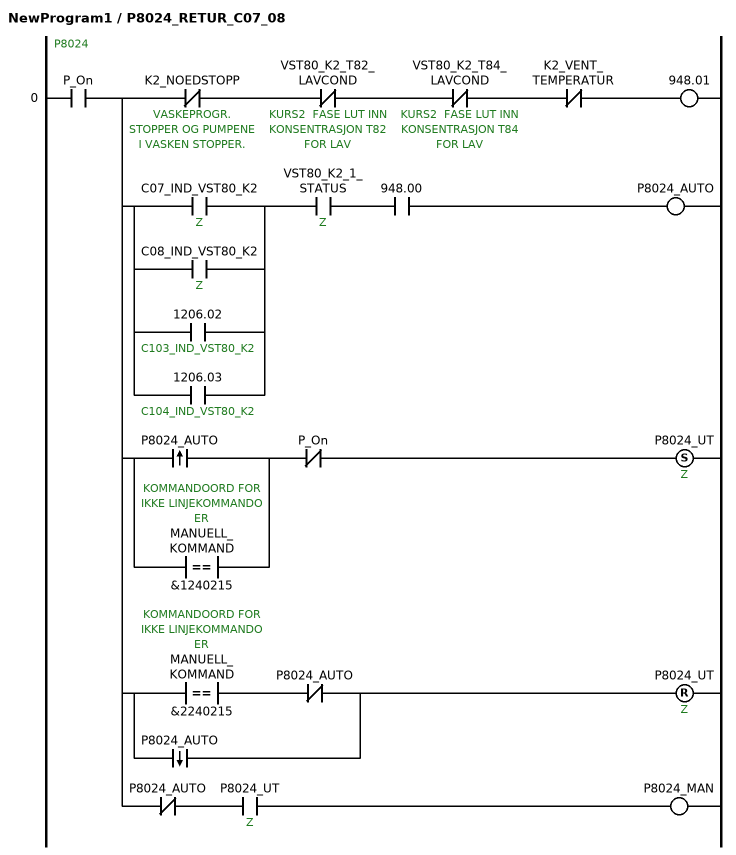
; rung 0: P8024
LD P_On
OUT TR0
ANDNOT K2_NOEDSTOPP  ; VASKEPROGR. STOPPER OG PUMPENE I VASKEN STOPPER.
ANDNOT VST80_K2_T82_LAVCOND  ; KURS2  FASE LUT INN KONSENTRASJON T82 FOR LAV
ANDNOT VST80_K2_T84_LAVCOND  ; KURS2  FASE LUT INN KONSENTRASJON T84 FOR LAV
ANDNOT K2_VENT_TEMPERATUR
OUT 948.01
LD TR0
LD C07_IND_VST80_K2  ; Z
OR C08_IND_VST80_K2  ; Z
OR 1206.02  ; C103_IND_VST80_K2
OR 1206.03  ; C104_IND_VST80_K2
ANDLD
AND VST80_K2_1_STATUS  ; Z
AND 948.00
OUT P8024_AUTO
LD TR0
@LD P8024_AUTO
OR=L(301) MANUELL_KOMMAND &1240215  ; KOMMANDOORD FOR IKKE LINJEKOMMANDOER
ANDLD
ANDNOT P_On
SET P8024_UT  ; Z
LD TR0
LD=L(301) MANUELL_KOMMAND &2240215  ; KOMMANDOORD FOR IKKE LINJEKOMMANDOER
ANDNOT P8024_AUTO
%OR P8024_AUTO
ANDLD
RSET P8024_UT  ; Z
LD TR0
ANDNOT P8024_AUTO
AND P8024_UT  ; Z
OUT P8024_MAN

### Section T40_TEMP_NIVÅ

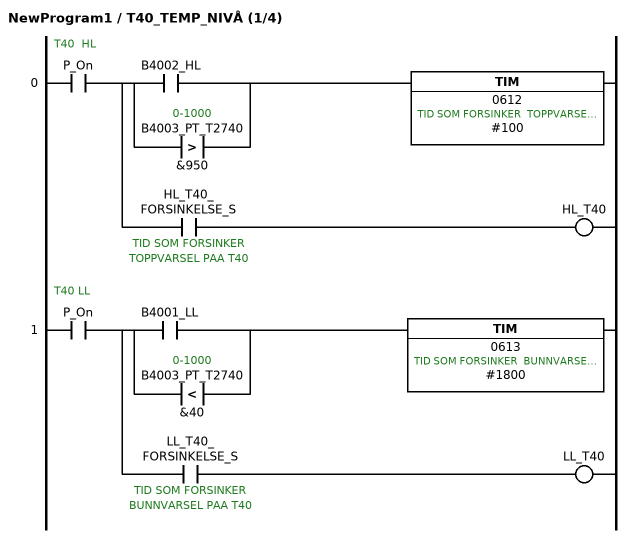
; rung 0: T40  HL
LD P_On
OUT TR0
LD B4002_HL
OR>(320) B4003_PT_T2740 &950  ; 0-1000
ANDLD
TIM 0612 #100  ; TID SOM FORSINKER  TOPPVARSEL PAA T40
LD TR0
AND HL_T40_FORSINKELSE_S  ; TID SOM FORSINKER  TOPPVARSEL PAA T40
OUT HL_T40
; rung 1: T40 LL
LD P_On
OUT TR0
LD B4001_LL
OR<(310) B4003_PT_T2740 &40  ; 0-1000
ANDLD
TIM 0613 #1800  ; TID SOM FORSINKER  BUNNVARSEL PAA T40
LD TR0
AND LL_T40_FORSINKELSE_S  ; TID SOM FORSINKER  BUNNVARSEL PAA T40
OUT LL_T40

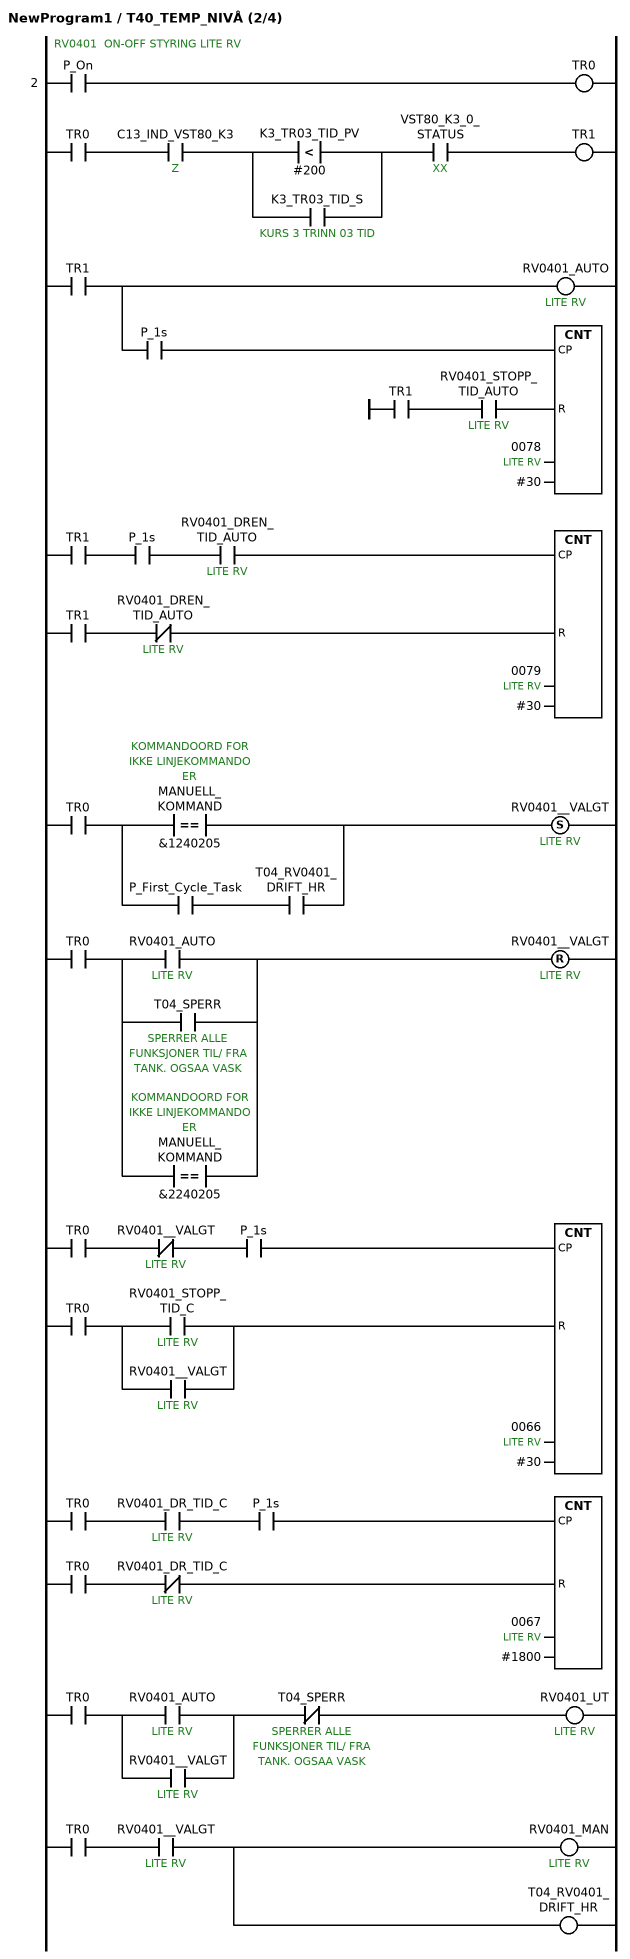
; rung 2: RV0401  ON-OFF STYRING LITE RV
LD P_On
OUT TR0
AND C13_IND_VST80_K3  ; Z
LD<(310) K3_TR03_TID_PV #200
OR K3_TR03_TID_S  ; KURS 3 TRINN 03 TID
ANDLD
AND VST80_K3_0_STATUS  ; XX
OUT TR1
OUT RV0401_AUTO  ; LITE RV
AND P_1s
LD TR1
AND RV0401_STOPP_TID_AUTO  ; LITE RV
CNT 0078 #30  ; LITE RV
LD TR1
AND P_1s
AND RV0401_DREN_TID_AUTO  ; LITE RV
LD TR1
ANDNOT RV0401_DREN_TID_AUTO  ; LITE RV
CNT 0079 #30  ; LITE RV
LD TR0
LD=L(301) MANUELL_KOMMAND &1240205  ; KOMMANDOORD FOR IKKE LINJEKOMMANDOER
LD P_First_Cycle_Task
AND T04_RV0401_DRIFT_HR
ORLD
ANDLD
SET RV0401__VALGT  ; LITE RV
LD TR0
LD RV0401_AUTO  ; LITE RV
OR T04_SPERR  ; SPERRER ALLE FUNKSJONER TIL/ FRA TANK. OGSAA VASK
OR=L(301) MANUELL_KOMMAND &2240205  ; KOMMANDOORD FOR IKKE LINJEKOMMANDOER
ANDLD
RSET RV0401__VALGT  ; LITE RV
LD TR0
ANDNOT RV0401__VALGT  ; LITE RV
AND P_1s
LD TR0
LD RV0401_STOPP_TID_C  ; LITE RV
OR RV0401__VALGT  ; LITE RV
ANDLD
CNT 0066 #30  ; LITE RV
LD TR0
AND RV0401_DR_TID_C  ; LITE RV
AND P_1s
LD TR0
ANDNOT RV0401_DR_TID_C  ; LITE RV
CNT 0067 #1800  ; LITE RV
LD TR0
LD RV0401_AUTO  ; LITE RV
OR RV0401__VALGT  ; LITE RV
ANDLD
ANDNOT T04_SPERR  ; SPERRER ALLE FUNKSJONER TIL/ FRA TANK. OGSAA VASK
OUT RV0401_UT  ; LITE RV
LD TR0
AND RV0401__VALGT  ; LITE RV
OUT RV0401_MAN  ; LITE RV
OUT T04_RV0401_DRIFT_HR

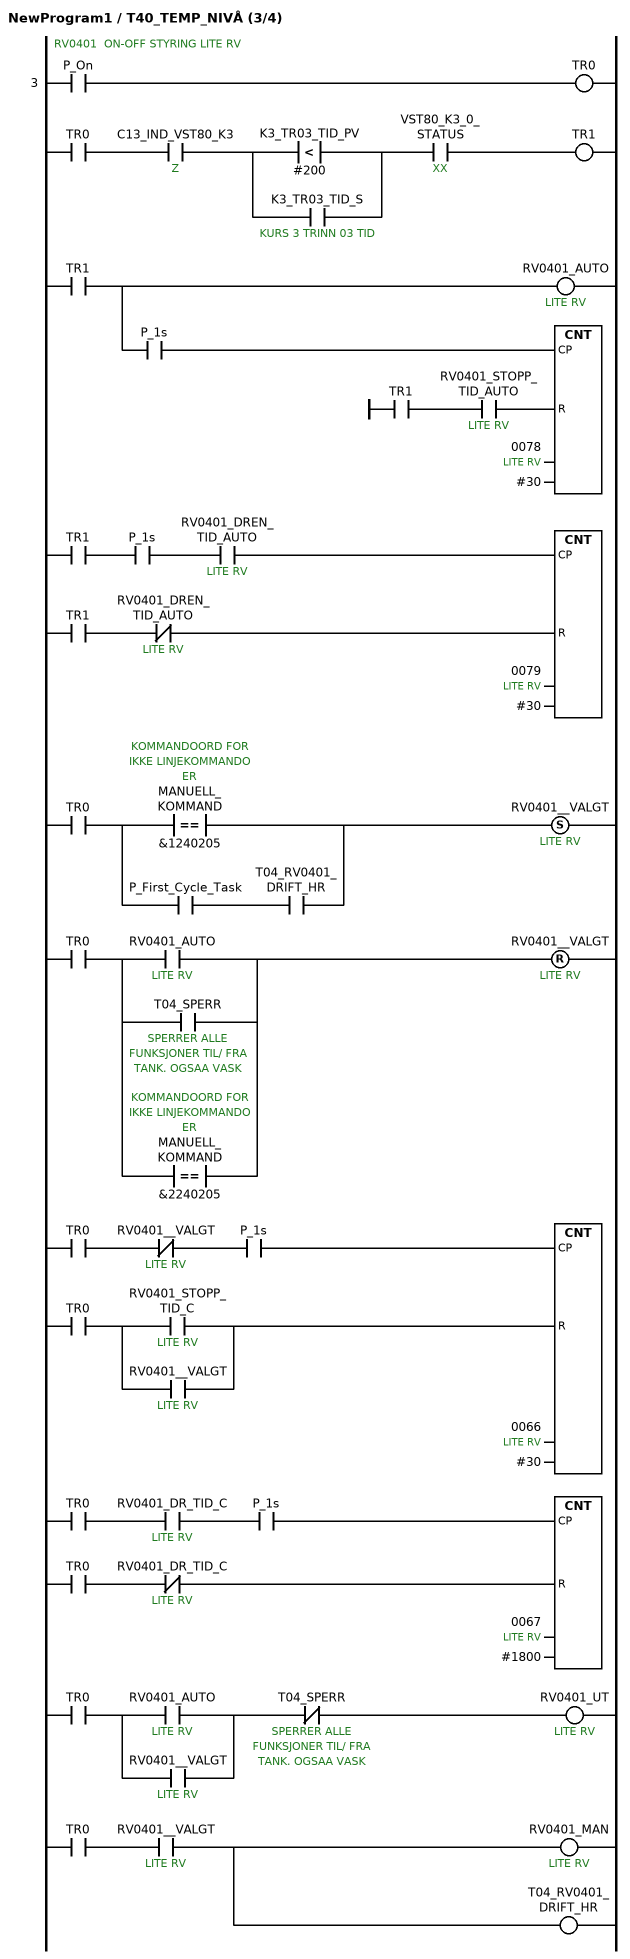
; rung 3: RV0401  ON-OFF STYRING LITE RV
LD P_On
OUT TR0
AND C13_IND_VST80_K3  ; Z
LD<(310) K3_TR03_TID_PV #200
OR K3_TR03_TID_S  ; KURS 3 TRINN 03 TID
ANDLD
AND VST80_K3_0_STATUS  ; XX
OUT TR1
OUT RV0401_AUTO  ; LITE RV
AND P_1s
LD TR1
AND RV0401_STOPP_TID_AUTO  ; LITE RV
CNT 0078 #30  ; LITE RV
LD TR1
AND P_1s
AND RV0401_DREN_TID_AUTO  ; LITE RV
LD TR1
ANDNOT RV0401_DREN_TID_AUTO  ; LITE RV
CNT 0079 #30  ; LITE RV
LD TR0
LD=L(301) MANUELL_KOMMAND &1240205  ; KOMMANDOORD FOR IKKE LINJEKOMMANDOER
LD P_First_Cycle_Task
AND T04_RV0401_DRIFT_HR
ORLD
ANDLD
SET RV0401__VALGT  ; LITE RV
LD TR0
LD RV0401_AUTO  ; LITE RV
OR T04_SPERR  ; SPERRER ALLE FUNKSJONER TIL/ FRA TANK. OGSAA VASK
OR=L(301) MANUELL_KOMMAND &2240205  ; KOMMANDOORD FOR IKKE LINJEKOMMANDOER
ANDLD
RSET RV0401__VALGT  ; LITE RV
LD TR0
ANDNOT RV0401__VALGT  ; LITE RV
AND P_1s
LD TR0
LD RV0401_STOPP_TID_C  ; LITE RV
OR RV0401__VALGT  ; LITE RV
ANDLD
CNT 0066 #30  ; LITE RV
LD TR0
AND RV0401_DR_TID_C  ; LITE RV
AND P_1s
LD TR0
ANDNOT RV0401_DR_TID_C  ; LITE RV
CNT 0067 #1800  ; LITE RV
LD TR0
LD RV0401_AUTO  ; LITE RV
OR RV0401__VALGT  ; LITE RV
ANDLD
ANDNOT T04_SPERR  ; SPERRER ALLE FUNKSJONER TIL/ FRA TANK. OGSAA VASK
OUT RV0401_UT  ; LITE RV
LD TR0
AND RV0401__VALGT  ; LITE RV
OUT RV0401_MAN  ; LITE RV
OUT T04_RV0401_DRIFT_HR

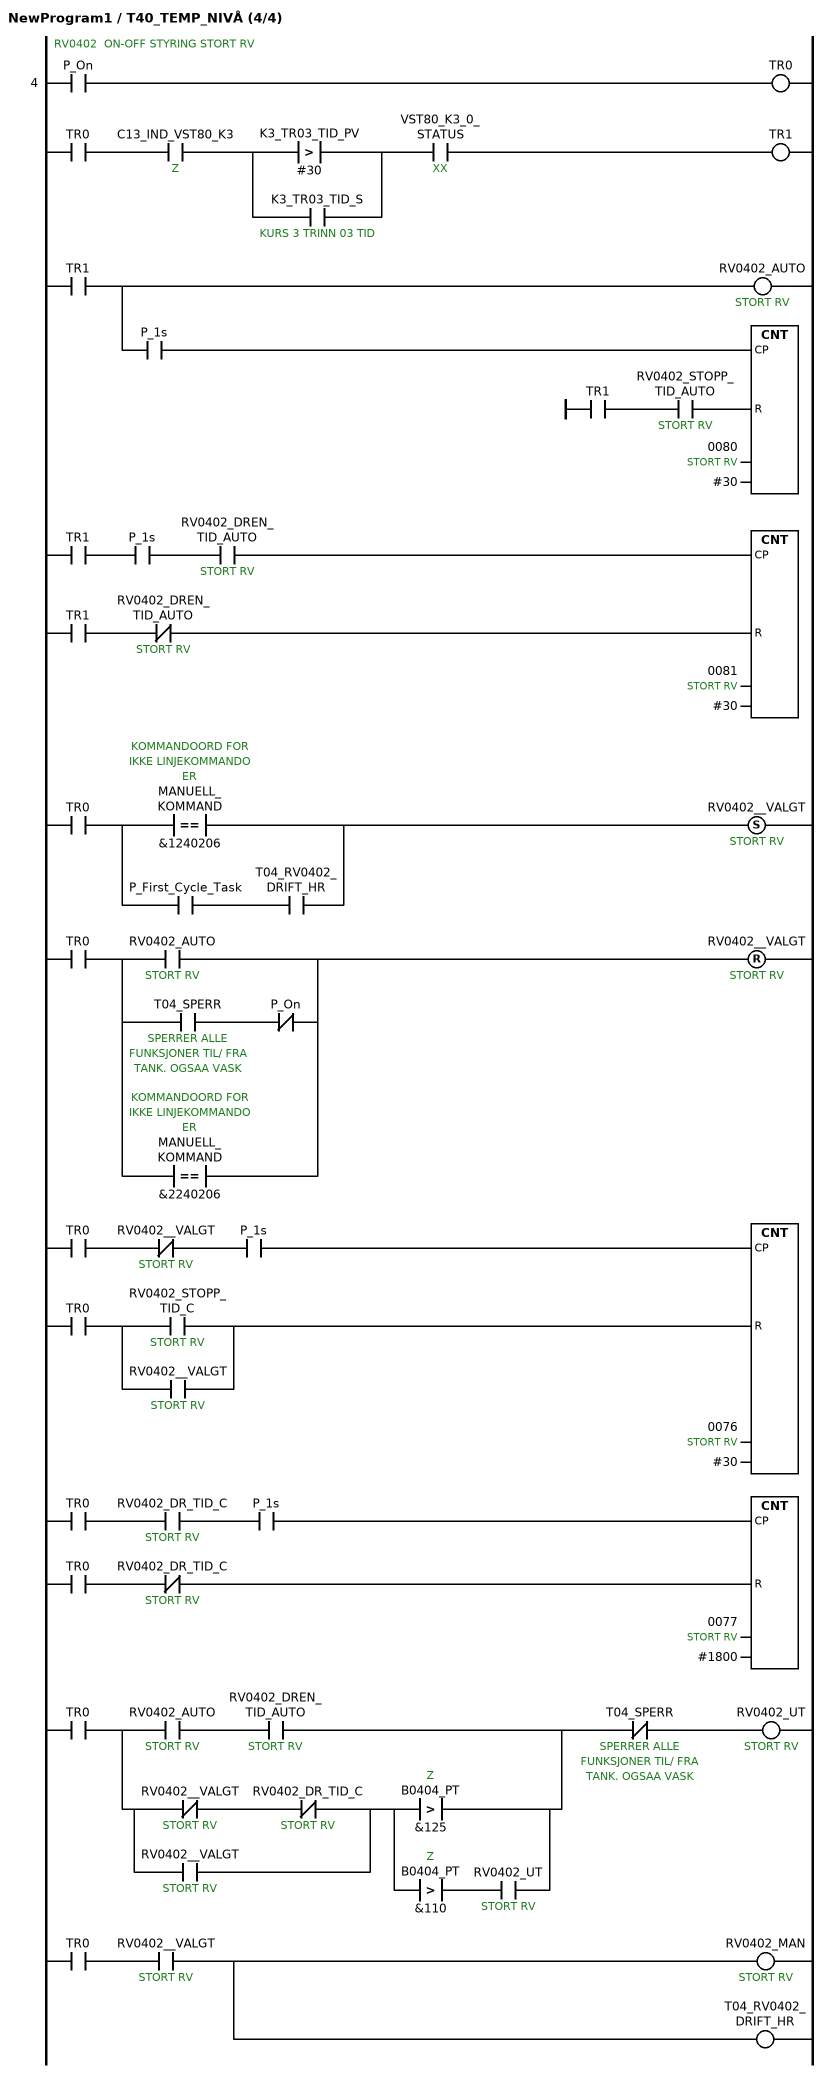
; rung 4: RV0402  ON-OFF STYRING STORT RV
LD P_On
OUT TR0
AND C13_IND_VST80_K3  ; Z
LD>(320) K3_TR03_TID_PV #30
OR K3_TR03_TID_S  ; KURS 3 TRINN 03 TID
ANDLD
AND VST80_K3_0_STATUS  ; XX
OUT TR1
OUT RV0402_AUTO  ; STORT RV
AND P_1s
LD TR1
AND RV0402_STOPP_TID_AUTO  ; STORT RV
CNT 0080 #30  ; STORT RV
LD TR1
AND P_1s
AND RV0402_DREN_TID_AUTO  ; STORT RV
LD TR1
ANDNOT RV0402_DREN_TID_AUTO  ; STORT RV
CNT 0081 #30  ; STORT RV
LD TR0
LD=L(301) MANUELL_KOMMAND &1240206  ; KOMMANDOORD FOR IKKE LINJEKOMMANDOER
LD P_First_Cycle_Task
AND T04_RV0402_DRIFT_HR
ORLD
ANDLD
SET RV0402__VALGT  ; STORT RV
LD TR0
LD RV0402_AUTO  ; STORT RV
LD T04_SPERR  ; SPERRER ALLE FUNKSJONER TIL/ FRA TANK. OGSAA VASK
ANDNOT P_On
ORLD
OR=L(301) MANUELL_KOMMAND &2240206  ; KOMMANDOORD FOR IKKE LINJEKOMMANDOER
ANDLD
RSET RV0402__VALGT  ; STORT RV
LD TR0
ANDNOT RV0402__VALGT  ; STORT RV
AND P_1s
LD TR0
LD RV0402_STOPP_TID_C  ; STORT RV
OR RV0402__VALGT  ; STORT RV
ANDLD
CNT 0076 #30  ; STORT RV
LD TR0
AND RV0402_DR_TID_C  ; STORT RV
AND P_1s
LD TR0
ANDNOT RV0402_DR_TID_C  ; STORT RV
CNT 0077 #1800  ; STORT RV
LD TR0
LD RV0402_AUTO  ; STORT RV
AND RV0402_DREN_TID_AUTO  ; STORT RV
LDNOT RV0402__VALGT  ; STORT RV
ANDNOT RV0402_DR_TID_C  ; STORT RV
OR RV0402__VALGT  ; STORT RV
LD>(320) B0404_PT &125  ; Z
LD>(320) B0404_PT &110  ; Z
AND RV0402_UT  ; STORT RV
ORLD
ANDLD
ORLD
ANDLD
ANDNOT T04_SPERR  ; SPERRER ALLE FUNKSJONER TIL/ FRA TANK. OGSAA VASK
OUT RV0402_UT  ; STORT RV
LD TR0
AND RV0402__VALGT  ; STORT RV
OUT RV0402_MAN  ; STORT RV
OUT T04_RV0402_DRIFT_HR

### Section T40_STATUS

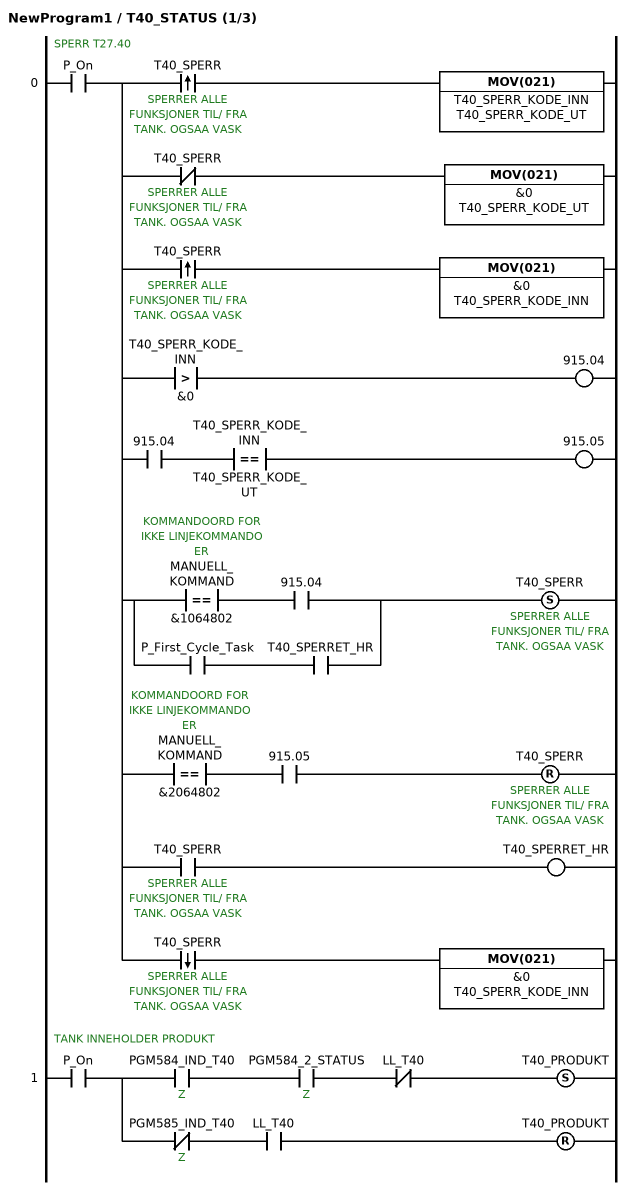
; rung 0: SPERR T27.40
LD P_On
OUT TR0
@AND T40_SPERR  ; SPERRER ALLE FUNKSJONER TIL/ FRA TANK. OGSAA VASK
MOV(021) T40_SPERR_KODE_INN T40_SPERR_KODE_UT
LD TR0
ANDNOT T40_SPERR  ; SPERRER ALLE FUNKSJONER TIL/ FRA TANK. OGSAA VASK
MOV(021) &0 T40_SPERR_KODE_UT
LD TR0
@AND T40_SPERR  ; SPERRER ALLE FUNKSJONER TIL/ FRA TANK. OGSAA VASK
MOV(021) &0 T40_SPERR_KODE_INN
LD TR0
AND>(320) T40_SPERR_KODE_INN &0
OUT 915.04
LD TR0
AND 915.04
AND=(300) T40_SPERR_KODE_INN T40_SPERR_KODE_UT
OUT 915.05
LD TR0
LD=L(301) MANUELL_KOMMAND &1064802  ; KOMMANDOORD FOR IKKE LINJEKOMMANDOER
AND 915.04
LD P_First_Cycle_Task
AND T40_SPERRET_HR
ORLD
ANDLD
SET T40_SPERR  ; SPERRER ALLE FUNKSJONER TIL/ FRA TANK. OGSAA VASK
LD TR0
AND=L(301) MANUELL_KOMMAND &2064802  ; KOMMANDOORD FOR IKKE LINJEKOMMANDOER
AND 915.05
RSET T40_SPERR  ; SPERRER ALLE FUNKSJONER TIL/ FRA TANK. OGSAA VASK
LD TR0
AND T40_SPERR  ; SPERRER ALLE FUNKSJONER TIL/ FRA TANK. OGSAA VASK
OUT T40_SPERRET_HR
LD TR0
%AND T40_SPERR  ; SPERRER ALLE FUNKSJONER TIL/ FRA TANK. OGSAA VASK
MOV(021) &0 T40_SPERR_KODE_INN
; rung 1: TANK INNEHOLDER PRODUKT
LD P_On
OUT TR0
AND PGM584_IND_T40  ; Z
AND PGM584_2_STATUS  ; Z
ANDNOT LL_T40
SET T40_PRODUKT
LD TR0
ANDNOT PGM585_IND_T40  ; Z
AND LL_T40
RSET T40_PRODUKT

